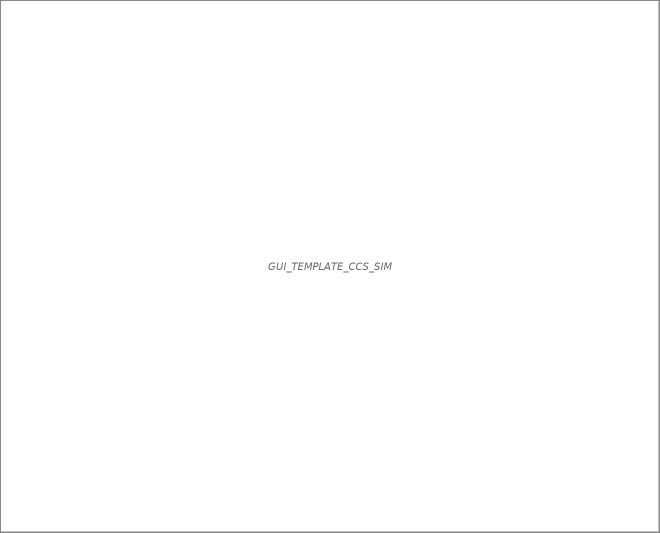
VISUALIZATION GUI_CCS_SIM  // 660x533
    Frame (0,0 660x533)
        shows GUI_TEMPLATE_CCS_SIM(m_DeviceName := ccssim, m_Instance := MAIN.ccs_sim)
END_VISUALIZATION

(* stored: Version 1.1.0.1, ProductVersion 3.1.4024.11
   Visu GUI_CCS_SIM: Id {b56db7a4-8ee3-4993-9130-35151cd4f7eb} *)
